PROGRAM MAIN
VAR
	bled1 AT %Q*: BOOL := FALSE;
	bsw1 AT %I*: BOOL := FALSE;
	bsw2 AT %I*: BOOL := FALSE;
	bled2 AT %Q*: BOOL := false;
END_VAR

bled1 := NOT bsw2;
bled2 := NOT bsw1;

END_PROGRAM

(* stored: Version 1.1.0.1, ProductVersion 3.1.4024.12
   POU MAIN: Id {7adc2b83-ae5d-4018-a640-34dc7c7d6846}, SpecialFunc None *)
